FUNCTION_BLOCK FB_Methods

(* Performs work on input data. *)
METHOD M_DoWork : BOOL
VAR_INPUT
    nStep : INT;
END_VAR
VAR_OUTPUT
    bOk : BOOL;
END_VAR
END_METHOD

END_FUNCTION_BLOCK

(* stored: Version 1.1.0.1
   POU FB_Methods: Id {11111111-1111-1111-1111-111111111103}
   Method M_DoWork: Id {22222222-2222-2222-2222-222222222201} *)
